/// Axis driver limit switch
FUNCTION_BLOCK FB_LimitSwitchRefSim
VAR_INPUT
	/// Aktiviert die Logik
	bEnable					:BOOL;
	/// Position der Achse
	fPosition				:REAL;
	
	/// Endschalter (Oeffner)
	bLimitSwitch			:BOOL;
	/// Distanz Simuliertem Ref-Schalter zu Endschalter
	fRefLimitDistance		:REAL := 1;
	
	/// Referenzposition
	fRefPosition			:REAL;
	/// Pruefen des Positionsbereichs der Referenzposition
	fRefPosCheckArea		:REAL := 0.2;
END_VAR
VAR_OUTPUT
	/// Endschalter (Verzeogert)
	bLimitSwitchSim			:BOOL;
	/// Simulierter Ref Schalter
	bRefSwitchSim			:BOOL;
	
	/// Pruefung der Refpos OK
	bRefCheckOk				:BOOL;
END_VAR
VAR
	
END_VAR
VAR PERSISTENT
	fPosLatched			:REAL;
	bPosLatched			:BOOL;
END_VAR

(*
	Baustein um einen Ref-Schalter und Limitswitch mit 1 Eingang zu realisieren
	RE / 2015 / www.rmth.at
*)

IF NOT bEnable THEN
	bLimitSwitchSim := bLimitSwitch;
	bRefSwitchSim := bLimitSwitchSim;
	bRefCheckOk := FALSE;
	RETURN;
END_IF

// logik
IF bLimitSwitch THEN // (Oeffner)
	fPosLatched := 0;
	bPosLatched := FALSE;	
	bLimitSwitchSim := TRUE; // limit ok
	bRefSwitchSim := FALSE; // kein referenz

ELSE
	// Position merken
	IF NOT bPosLatched THEN
		bPosLatched := TRUE;
		fPosLatched := fPosition;
	END_IF

	bRefSwitchSim := TRUE;
	bLimitSwitchSim := (ABS(fPosition - fPosLatched) >= fRefLimitDistance);
END_IF

// Referenzpunkt pruefen
bRefCheckOk := ABS(fRefPosition - fPosLatched) <= fRefPosCheckArea;

METHOD Reset : bool
VAR_INPUT
END_VAR
fPosLatched := 0;
bPosLatched := FALSE;
END_METHOD

END_FUNCTION_BLOCK

(* stored: Version 1.1.0.1, ProductVersion 3.1.4022.9
   POU FB_LimitSwitchRefSim: Id {48eb2f9c-6246-4468-a584-ccfc532dff24}, SpecialFunc None
   Method Reset: Id {b2907d14-785f-42e7-948f-44ba3218f996} *)
